Staubli VAL3: sendStatus.pgx

program sendStatus()
  local num buffer[79]
  local point currentPosition
  local joint currentPose
  local num moveId
begin
  buffer[0] = MAGIC_HEADER
  buffer[1] = 131

  currentPosition = here(endEffector, world)
  call encodePoint(currentPosition, buffer[2])

  currentPose = herej()
  call encodeJoint(currentPose, buffer[26])

  currentPose = getPositionErr()
  call encodeJoint(currentPose, buffer[50])

  buffer[74] = sel(isSettled(), 1, 0)

  moveId = getMoveId()
  toBinary(moveId, 1, "4.0b", buffer[75])

  sioSet(socket, buffer)
end
